INTERFACE I_ArrayDatatype_2D EXTENDS I_ArrayDatatype

METHOD PUBLIC TryGetElementAsDatatypeByIndex : BOOL
VAR_INPUT
	Index1 : DINT;
	Index2 : DINT;
	Destination : REFERENCE TO I_Datatype;
END_VAR
END_METHOD

END_INTERFACE

(* stored: Version 1.1.0.1, ProductVersion 3.1.4024.13
   Itf I_ArrayDatatype_2D: Id {45e50fe4-4fd7-047a-0e00-622e98d27408}
   Method TryGetElementAsDatatypeByIndex: Id {c4c34bb1-c48f-00a5-2950-d43a7880b3d5} *)
